FUNCTION_BLOCK FB_OperatorStation
VAR
    eState                    : E_OperatorExchangeState := E_OperatorExchangeState.Idle;
    eInstruction              : E_OperatorInstruction := E_OperatorInstruction.None;
    sMessage                  : STRING(255);
    stStatusInternal          : ST_OperatorStationStatus;

    bExchangeComplete         : BOOL;
    bPartRemovedConfirmed     : BOOL;
    bRejectConfirmed          : BOOL;
    bRejectArmed              : BOOL;
    bRejectEdgeAccepted       : BOOL;
    bPreviousRejectSensor     : BOOL;
    bRejectPulse              : BOOL;
    rtIndexAttempt : R_TRIG;
    bIndexAttemptActive : BOOL;
    bLoadSetComplete : BOOL;
    bLoadSetEmpty : BOOL;
    bMissingPbupAlert : BOOL;
    bMissingProductAlert : BOOL;
END_VAR

METHOD PUBLIC Cyclic
VAR_INPUT
    bAutomaticActive          : BOOL;
    bIndexStable              : BOOL;
    stOperatorNest            : ST_Nest;
    bPartPresent              : BOOL;
    bPbupPresent : BOOL;
    bTwoHandsSafe : BOOL;
    bResetRequest : BOOL;
    bRejectChutePartPresent   : BOOL;
    bRequireRejectConfirm     : BOOL;
    bAllowEmptyNestIndex      : BOOL;
END_VAR
// Product and PBUP form one load set; retain the legacy product/reject semantics.
bLoadSetComplete := bPartPresent AND bPbupPresent;
bLoadSetEmpty := NOT bPartPresent AND NOT bPbupPresent;
rtIndexAttempt(CLK := bTwoHandsSafe);
IF NOT bAutomaticActive OR NOT bTwoHandsSafe OR NOT bIndexStable OR bResetRequest THEN
    bIndexAttemptActive := FALSE;
ELSIF rtIndexAttempt.Q THEN
    bIndexAttemptActive := TRUE;
END_IF
IF NOT bAutomaticActive OR bResetRequest OR NOT (bPartPresent XOR bPbupPresent) THEN
    bMissingPbupAlert := FALSE;
    bMissingProductAlert := FALSE;
ELSIF bIndexAttemptActive THEN
    bMissingPbupAlert := bPartPresent AND NOT bPbupPresent;
    bMissingProductAlert := bPbupPresent AND NOT bPartPresent;
END_IF


bRejectPulse :=
    bRejectChutePartPresent
    AND NOT bPreviousRejectSensor;

bPreviousRejectSensor := bRejectChutePartPresent;
bRejectEdgeAccepted := FALSE;

IF NOT bAutomaticActive THEN

    eState := E_OperatorExchangeState.Idle;
    bExchangeComplete := FALSE;
    bPartRemovedConfirmed := FALSE;
    bRejectConfirmed := FALSE;
    bRejectArmed := FALSE;
    eInstruction := E_OperatorInstruction.None;
    sMessage := '';

ELSE

    CASE eState OF

        E_OperatorExchangeState.Idle:
            bExchangeComplete := FALSE;
            eInstruction := E_OperatorInstruction.None;
            sMessage := '';

            IF bIndexStable THEN
                eState := E_OperatorExchangeState.EvaluateNest;
            END_IF

        E_OperatorExchangeState.EvaluateNest:
            bExchangeComplete := FALSE;
            bPartRemovedConfirmed := FALSE;
            bRejectConfirmed := FALSE;
            bRejectArmed := FALSE;

            IF stOperatorNest.stResult.bValid
				OR (stOperatorNest.eDisposition = E_PartDisposition.Reprocess)
			THEN

                IF bPartPresent THEN
                    eState := E_OperatorExchangeState.WaitingForPartRemoval;
                ELSE
                    bPartRemovedConfirmed := TRUE;

					IF (stOperatorNest.eDisposition <> E_PartDisposition.Reprocess)
						AND NOT stOperatorNest.stResult.bPassed
						AND bRequireRejectConfirm
					THEN
                        eState := E_OperatorExchangeState.WaitingForRejectConfirmation;
                    ELSE
                        eState := E_OperatorExchangeState.WaitingForPartLoading;
                    END_IF
                END_IF

            ELSE
                eState := E_OperatorExchangeState.WaitingForPartLoading;
            END_IF

        E_OperatorExchangeState.WaitingForPartRemoval:

            IF stOperatorNest.eDisposition = E_PartDisposition.Reprocess THEN

				// Reprocess is neither PASS nor definitive FAIL.
				// The operator must remove the part, but it must NOT
				// be sent to the reject chute.
				eInstruction :=
					E_OperatorInstruction.RemoveFailedPart;
			
				sMessage :=
					'Remove part for reprocess';
			
			ELSIF stOperatorNest.stResult.bPassed THEN
			
				eInstruction :=
					E_OperatorInstruction.RemovePassedPart;
			
				sMessage :=
					'Remove passed part from operator nest';
			
			ELSE
			
				eInstruction :=
					E_OperatorInstruction.RemoveFailedPart;
			
				sMessage :=
					'Remove failed part from operator nest';
			
			END_IF

            IF NOT bPartPresent THEN
                bPartRemovedConfirmed := TRUE;
                bRejectArmed := FALSE;

				IF (stOperatorNest.eDisposition = E_PartDisposition.Reprocess) THEN
				
					// Reprocess parts must NOT go to the reject chute.
					eState :=
						E_OperatorExchangeState.WaitingForPartLoading;
				
				ELSIF NOT stOperatorNest.stResult.bPassed
					AND bRequireRejectConfirm
				THEN
				
					eState :=
						E_OperatorExchangeState.WaitingForRejectConfirmation;
				
				ELSE
				
					eState :=
						E_OperatorExchangeState.WaitingForPartLoading;
				
				END_IF
            END_IF

        E_OperatorExchangeState.WaitingForRejectConfirmation:

            eInstruction := E_OperatorInstruction.PlacePartInRejectBin;

            IF NOT bRejectChutePartPresent THEN
                bRejectArmed := TRUE;
            END_IF

            IF NOT bRejectArmed THEN
                sMessage := 'Clear reject chute, then place the failed part into reject chute';
            ELSE
                sMessage := 'Place failed part into reject chute';
            END_IF

            IF bPartRemovedConfirmed
                AND bRejectArmed
                AND bRejectPulse
            THEN
                bRejectConfirmed := TRUE;
                bRejectEdgeAccepted := TRUE;
            END_IF

            IF bPartRemovedConfirmed
                AND bRejectConfirmed
            THEN
                eState := E_OperatorExchangeState.WaitingForPartLoading;
            END_IF

        E_OperatorExchangeState.WaitingForPartLoading:
            bExchangeComplete := FALSE;
            eInstruction := E_OperatorInstruction.LoadPart;
            IF bLoadSetComplete THEN
                eInstruction := E_OperatorInstruction.ReadyToIndex;
                sMessage := 'Product and PBUP loaded - press two-hand buttons to index';
                bExchangeComplete := TRUE;
                eState := E_OperatorExchangeState.ExchangeComplete;
            ELSIF bLoadSetEmpty AND bAllowEmptyNestIndex THEN
                eInstruction := E_OperatorInstruction.ReadyToIndexEmpty;
                sMessage := 'Load product and PBUP or continue with empty nest';
                bExchangeComplete := TRUE;
                eState := E_OperatorExchangeState.ExchangeComplete;
            ELSIF bPartPresent THEN
                sMessage := 'PBUP missing - load PBUP or remove product';
            ELSIF bPbupPresent THEN
                sMessage := 'Product missing - load product or remove PBUP';
            ELSE
                sMessage := 'Load product and PBUP into operator nest';
            END_IF

        E_OperatorExchangeState.ExchangeComplete:
            // Never use a latched exchange completion to permit a later partial load.
            IF NOT bIndexStable THEN
                eState := E_OperatorExchangeState.WaitingForTableIndexComplete;
            ELSIF bLoadSetComplete THEN
                bExchangeComplete := TRUE;
                eInstruction := E_OperatorInstruction.ReadyToIndex;
                sMessage := 'Product and PBUP loaded - press two-hand buttons to index';
            ELSIF bLoadSetEmpty AND bAllowEmptyNestIndex THEN
                bExchangeComplete := TRUE;
                eInstruction := E_OperatorInstruction.ReadyToIndexEmpty;
                sMessage := 'Empty nest - press two-hand buttons to index';
            ELSE
                bExchangeComplete := FALSE;
                eState := E_OperatorExchangeState.WaitingForPartLoading;
                eInstruction := E_OperatorInstruction.LoadPart;
                IF bPartPresent THEN
                    sMessage := 'PBUP missing - load PBUP or remove product';
                ELSIF bPbupPresent THEN
                    sMessage := 'Product missing - load product or remove PBUP';
                ELSE
                    sMessage := 'Load product and PBUP into operator nest';
                END_IF
            END_IF

        E_OperatorExchangeState.WaitingForTableIndexComplete:

            eInstruction := E_OperatorInstruction.TableIndexing;
            sMessage := 'Table index in progress';

            IF bIndexStable THEN
                bExchangeComplete := FALSE;
                bPartRemovedConfirmed := FALSE;
                bRejectConfirmed := FALSE;
                bRejectArmed := FALSE;
                eState := E_OperatorExchangeState.EvaluateNest;
            END_IF

        E_OperatorExchangeState.Fault:
            bExchangeComplete := FALSE;
            eInstruction := E_OperatorInstruction.None;
            sMessage := 'Operator exchange fault';

    END_CASE
END_IF

stStatusInternal.eState := eState;
stStatusInternal.eInstruction := eInstruction;

stStatusInternal.bExchangeComplete := bExchangeComplete;

stStatusInternal.bIndexPermissive :=
    bExchangeComplete
    AND eState = E_OperatorExchangeState.ExchangeComplete
    AND (bLoadSetComplete OR (bLoadSetEmpty AND bAllowEmptyNestIndex));

stStatusInternal.bPartRemovedConfirmed := bPartRemovedConfirmed;
stStatusInternal.bRejectConfirmed := bRejectConfirmed;
stStatusInternal.bRejectArmed := bRejectArmed;
stStatusInternal.bRejectEdgeAccepted := bRejectEdgeAccepted;

stStatusInternal.bRejectWaitingForClear :=
    (eState = E_OperatorExchangeState.WaitingForRejectConfirmation)
    AND NOT bRejectArmed;

stStatusInternal.bRejectPopupRequest :=
    (
        eState = E_OperatorExchangeState.WaitingForPartRemoval
        AND (stOperatorNest.eDisposition <> E_PartDisposition.Reprocess)
        AND stOperatorNest.stResult.bValid
        AND NOT stOperatorNest.stResult.bPassed
    )
    OR
    (
        eState = E_OperatorExchangeState.WaitingForRejectConfirmation
        AND (stOperatorNest.eDisposition <> E_PartDisposition.Reprocess)
    );

stStatusInternal.bPartPresent := bPartPresent;
stStatusInternal.bRejectChutePartPresent := bRejectChutePartPresent;
stStatusInternal.bResultValid := stOperatorNest.stResult.bValid;
stStatusInternal.bResultPassed := stOperatorNest.stResult.bPassed;
stStatusInternal.sMessage := sMessage;







stStatusInternal.bPbupPresent := bPbupPresent;
stStatusInternal.bLoadSetComplete := bLoadSetComplete;
stStatusInternal.bMissingPbup := bPartPresent AND NOT bPbupPresent;
stStatusInternal.bMissingProduct := bPbupPresent AND NOT bPartPresent;
stStatusInternal.bMissingPbupAlert := bMissingPbupAlert;
stStatusInternal.bMissingProductAlert := bMissingProductAlert;
END_METHOD

METHOD PUBLIC GetInstruction : E_OperatorInstruction
GetInstruction := eInstruction;
END_METHOD

METHOD PUBLIC GetState : E_OperatorExchangeState
GetState := eState;
END_METHOD

METHOD PUBLIC GetStatus : ST_OperatorStationStatus
GetStatus := stStatusInternal;
END_METHOD

METHOD PUBLIC IndexPermissive : BOOL
IndexPermissive := stStatusInternal.bIndexPermissive;
END_METHOD

METHOD PUBLIC IsComplete : BOOL
IsComplete := bExchangeComplete;
END_METHOD

END_FUNCTION_BLOCK

(* stored: Version 1.1.0.1, ProductVersion 3.1.4026.18
   POU FB_OperatorStation: Id {ff731f13-9fb1-43b6-a19e-d679d0a53809}, SpecialFunc None
   Method Cyclic: Id {511ffeea-7deb-4d8b-b22e-31cebd596b3a}
   Method GetInstruction: Id {96151fe5-6551-4687-9395-251188bc16e1}
   Method GetState: Id {50b48489-931c-45af-9267-a204b226aafd}
   Method GetStatus: Id {e74991c2-1064-4f40-b23e-9f8304b38600}
   Method IndexPermissive: Id {73d11cbf-354c-424e-a2a8-318ace7b680f}
   Method IsComplete: Id {44a76064-7b6e-440a-b915-9333a5f0a70e} *)
